// Mitsubishi GX Works2 project: 15dan   PLC: Q03UDV

PROGRAM MAIN
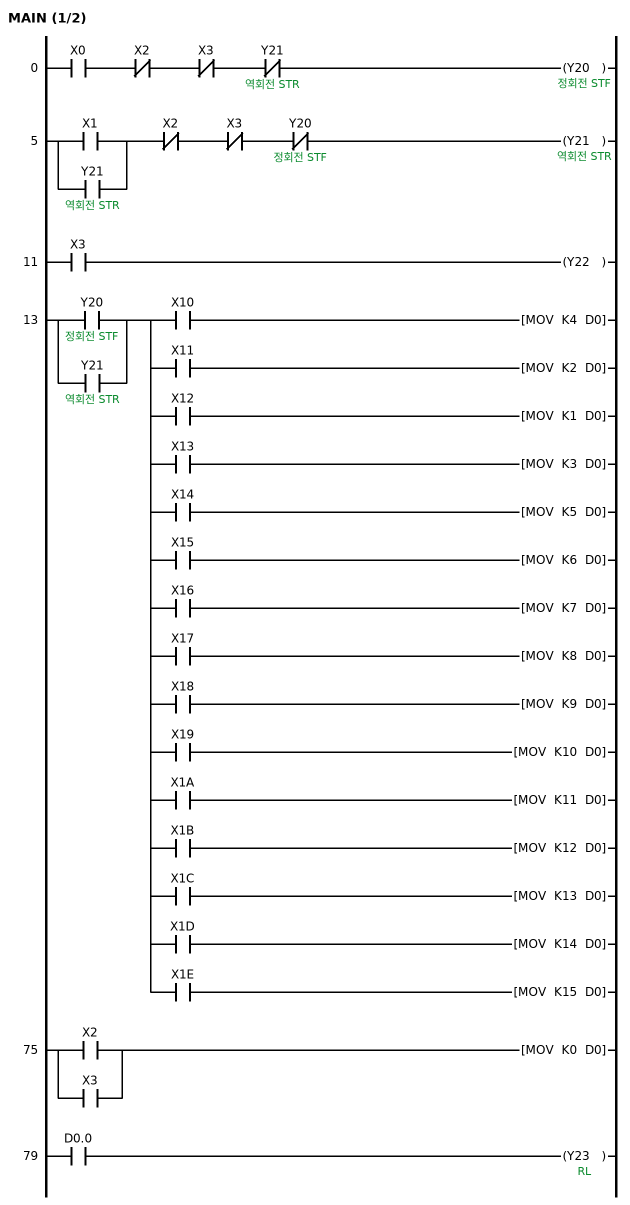
0     LD      X0
      ANI     X2
      ANI     X3
      ANI     Y21  ; 역회전 STR
      OUT     Y20  ; 정회전 STF
5     LD      X1
      OR      Y21  ; 역회전 STR
      ANI     X2
      ANI     X3
      ANI     Y20  ; 정회전 STF
      OUT     Y21  ; 역회전 STR
11    LD      X3
      OUT     Y22
13    LD      Y20  ; 정회전 STF
      OR      Y21  ; 역회전 STR
      MPS
      AND     X10
      MOV     K4 D0
      MRD
      AND     X11
      MOV     K2 D0
      MRD
      AND     X12
      MOV     K1 D0
      MRD
      AND     X13
      MOV     K3 D0
      MRD
      AND     X14
      MOV     K5 D0
      MRD
      AND     X15
      MOV     K6 D0
      MRD
      AND     X16
      MOV     K7 D0
      MRD
      AND     X17
      MOV     K8 D0
      MRD
      AND     X18
      MOV     K9 D0
      MRD
      AND     X19
      MOV     K10 D0
      MRD
      AND     X1A
      MOV     K11 D0
      MRD
      AND     X1B
      MOV     K12 D0
      MRD
      AND     X1C
      MOV     K13 D0
      MRD
      AND     X1D
      MOV     K14 D0
      MPP
      AND     X1E
      MOV     K15 D0
75    LD      X2
      OR      X3
      MOV     K0 D0
79    LD      D0.0
      OUT     Y23  ; RL
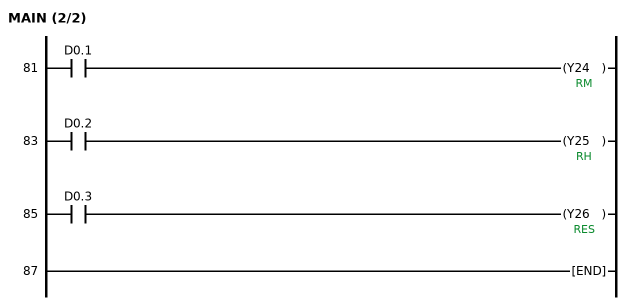
81    LD      D0.1
      OUT     Y24  ; RM
83    LD      D0.2
      OUT     Y25  ; RH
85    LD      D0.3
      OUT     Y26  ; RES
87    END
END_PROGRAM

PROGRAM speedBit
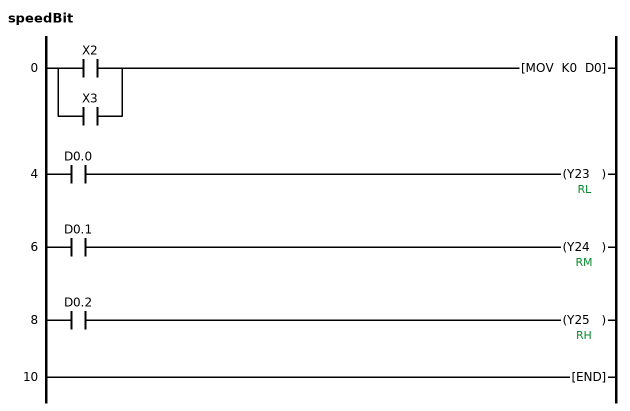
0     LD      X2
      OR      X3
      MOV     K0 D0
4     LD      D0.0
      OUT     Y23  ; RL
6     LD      D0.1
      OUT     Y24  ; RM
8     LD      D0.2
      OUT     Y25  ; RH
10    END
END_PROGRAM
